FUNCTION TryConvert_UDINT_TO_TOD : BOOL
VAR_INPUT
	in : UDINT;
	out : REFERENCE TO TOD;
END_VAR

IF in > DatatypeLimits.MAX_VALUE_OF_UDINT_WHICH_CAN_BE_HELD_IN_A_TOD THEN
	RETURN;
END_IF

out := UDINT_TO_TOD(in);
TryConvert_UDINT_TO_TOD := TRUE;

END_FUNCTION

(* stored: Version 1.1.0.1, ProductVersion 3.1.4024.12
   POU TryConvert_UDINT_TO_TOD: Id {ecddae14-fedb-4df5-9b15-cd779d6e1dcb}, SpecialFunc None *)
